TYPE Soft_Event_Control :
STRUCT
	Soft_Event_0 : BIT;
	Soft_Event_1 : BIT;
	Soft_Event_2 : BIT;
	Soft_Event_3 : BIT;
	Soft_Event_4 : BIT;
	Soft_Event_5 : BIT;
	Soft_Event_6 : BIT;
	Soft_Event_7 : BIT;
END_STRUCT
END_TYPE

(* stored: Version 1.1.0.1, ProductVersion 3.1.4024.10
   DUT Soft_Event_Control: Id {96123580-3c07-4592-90dd-5bd4424f2a50} *)
